FUNCTION_BLOCK FB_Fahrleitsystem
VAR_INPUT
END_VAR
VAR_OUTPUT
END_VAR
VAR
	Done : BOOL;
	Busy	: BOOL;
	Error : BOOL;
	StartStockwerk:	INT;
	ZielStockwerk:	INT;
	SicherheitsCheckbestanden : BOOL;
	AmStartStockwerk : BOOL;
	AmZielStockwerk : BOOL;
	TuerenZu : BOOL;
	Start : BOOL;
	AktuellesStockwerk : INT;
	Fahrauftragverstanden : BOOL;
	Tuerauftragverstanden : BOOL;
	State: ENUM_Fahrsystem;
	fbTuer : FB_Tuer;
	fbAchse : FB_Achse;
	AbholungFertig : BOOL;
	Closingdoors: BOOL;
	Achsereferenziert: BOOL;
	AufstartenAbgeschlossen : BOOL;
	AufstartenFreigabe : BOOL;
	AllDoorsClosed : BOOL;
	fbBlinker : FB_Blinker;
	FehlerQuittierenFlanke : R_TRIG;   // NEU — Flanke für Quittierung
 	sFehlertext : STRING(500);  // lokale Hilfsvariable
    i_txt       : INT;
END_VAR

fbAchse(Simulation:= , S_Zielposition:= , Achse:= IO_L1.LiftAxis);
fbTuer(
    SensorOpen1 := IO_L1.Door_1_SensorOpen,
    SensorOpen2 := IO_L1.Door_2_SensorOpen,
    SensorOpen3 := IO_L1.Door_3_SensorOpen,
    SensorOpen4 := IO_L1.Door_4_SensorOpen,
    SensorOpen5 := IO_L1.Door_5_SensorOpen,
    SensorOpen6 := IO_L1.Door_6_SensorOpen,

    SensorClosed1 := IO_L1.Door_1_SensorClosed,
    SensorClosed2 := IO_L1.Door_2_SensorClosed,
    SensorClosed3 := IO_L1.Door_3_SensorClosed,
    SensorClosed4 := IO_L1.Door_4_SensorClosed,
    SensorClosed5 := IO_L1.Door_5_SensorClosed,
    SensorClosed6 := IO_L1.Door_6_SensorClosed,

    Lichtschranke1 := IO_L1.Door_1_SensorActive,
    Lichtschranke2 := IO_L1.Door_2_SensorActive,
    Lichtschranke3 := IO_L1.Door_3_SensorActive,
    Lichtschranke4 := IO_L1.Door_4_SensorActive,
    Lichtschranke5 := IO_L1.Door_5_SensorActive,
    Lichtschranke6 := IO_L1.Door_6_SensorActive,

    MotorOpen1 => IO_L1.Door_1_MotorOpen,
    MotorOpen2 => IO_L1.Door_2_MotorOpen,
    MotorOpen3 => IO_L1.Door_3_MotorOpen,
    MotorOpen4 => IO_L1.Door_4_MotorOpen,
    MotorOpen5 => IO_L1.Door_5_MotorOpen,
    MotorOpen6 => IO_L1.Door_6_MotorOpen,

    MotorClose1 => IO_L1.Door_1_MotorClose,
    MotorClose2 => IO_L1.Door_2_MotorClose,
    MotorClose3 => IO_L1.Door_3_MotorClose,
    MotorClose4 => IO_L1.Door_4_MotorClose,
    MotorClose5 => IO_L1.Door_5_MotorClose,
    MotorClose6 => IO_L1.Door_6_MotorClose,
	AllDoorsClosed => AllDoorsClosed,
	FehlerQuittieren := IO_L1.Control_Reset
);

fbBlinker(bEnable:= TRUE, tOn:= T#500MS, tOff:=T#500MS , bOut=> );
SicherheitsCheckbestanden := FALSE;
Done := FALSE;
CASE State OF


	ENUM_Fahrsystem.Warten:
		Busy := FALSE;
		Done := FALSE;
		IF NOT 	AufstartenAbgeschlossen  AND IO_L1.Control_Automatic THEN
			Busy := TRUE;
			State := ENUM_Fahrsystem.Aufstartablauf;
		END_IF
		IF Start AND Divers.AutomatikmodusAktiv THEN
			Busy := TRUE;
			Start := FALSE;
			State := ENUM_Fahrsystem.Sicherheitscheck;
		END_IF
 		IF Visu_Manuellmodus.PosAnfahren AND Divers.ManuellmodusAktiv THEN
			ZielStockwerk := Visu_Manuellmodus.Zielstock;
 			State := ENUM_Fahrsystem.ZumZielStockwerk; 
		END_IF
	ENUM_Fahrsystem.Sicherheitscheck:
		//IF fbTuer.M_AreDoorsClosed() AND NOT fbAchse.M_isBusy() AND NOT fbAchse.M_hasError() THEN
			SicherheitsCheckbestanden := TRUE;
		//END_IF
		IF SicherheitsCheckbestanden THEN
			IF StartStockwerk = AktuellesStockwerk THEN
				State := ENUM_Fahrsystem.ZumZielStockwerk;
			END_IF
			IF StartStockwerk <> AktuellesStockwerk THEN 
				State := ENUM_Fahrsystem.ZumStartStockwerk;
			END_IF
		END_IF
		
	ENUM_Fahrsystem.Tueren:
		Busy := TRUE;	
		IF NOT Tuerauftragverstanden AND NOT fbAchse.M_isBusy() AND NOT fbAchse.M_hasError()THEN
			Tuerauftragverstanden := fbTuer.M_Tuerablaufstarten(AktuellesStockwerk);
		END_IF
		IF fbTuer.M_DoorOpen() THEN
			AbholungFertig := TRUE;
		ELSE 
			AbholungFertig := FALSE;
		END_IF
		IF fbTuer.M_isDone() THEN
			AbholungFertig := FALSE;
			Tuerauftragverstanden := FALSE;
			IF AmStartStockwerk THEN
				State := ENUM_Fahrsystem.ZumZielStockwerk;
			END_IF
			IF AmZielStockwerk THEN
				Done := TRUE; 
				State := ENUM_Fahrsystem.Warten;
			END_IF
		END_IF
	ENUM_Fahrsystem.ZumStartStockwerk:
		Busy := TRUE;
		AmZielStockwerk := FALSE;
		Fahrauftragverstanden := fbAchse.M_Movetoposition(StartStockwerk);
		IF fbAchse.M_isDone() THEN
			//OrderID_Counter.AktuellesStockwerk := StartStockwerk;
			AktuellesStockwerk := StartStockwerk;
			AmStartStockwerk := TRUE;
			State := ENUM_Fahrsystem.Tueren;
		END_IF
	ENUM_Fahrsystem.ZumZielStockwerk:
		Busy := TRUE;
		AmStartStockwerk := FALSE;
		Fahrauftragverstanden := fbAchse.M_Movetoposition(ZielStockwerk);
		IF fbAchse.M_isDone() THEN
			//OrderID_Counter.AktuellesStockwerk := ZielStockwerk;
			AktuellesStockwerk := ZielStockwerk;
			AmZielStockwerk := TRUE;
			IF Divers.AutomatikmodusAktiv THEN
				State := ENUM_Fahrsystem.Tueren;
			ELSE
				State := ENUM_Fahrsystem.Warten;	
			END_IF
			
		END_IF
	
	ENUM_Fahrsystem.Aufstartablauf: 
	Busy := TRUE;
	IF IO_L1.Control_Start THEN
		AufstartenFreigabe := TRUE;
	END_IF
		IF AufstartenFreigabe THEN
	
			IF NOT AllDoorsClosed THEN
				IO_L1.Control_LED_White := TRUE;
				Closingdoors := fbTuer.M_closeAllDoors();
			END_IF
			IF AllDoorsClosed THEN
				IO_L1.Control_LED_Red := TRUE;
				Achsereferenziert := fbAchse.M_Movetoposition(1);
					IF fbAchse.M_isDone() THEN
						AktuellesStockwerk := 1;
						AufstartenAbgeschlossen := TRUE;
						AufstartenFreigabe := FALSE;
						State := ENUM_Fahrsystem.Warten;
				END_IF
			END_IF
			
		END_IF
		
END_CASE


//LED Stuerung
IF IO_L1.Control_Automatic AND AufstartenAbgeschlossen THEN
    // Anlage läuft (mit oder ohne Auftrag) → dauernd an
    IO_L1.Control_LED_White := TRUE;

ELSIF IO_L1.Control_Automatic AND NOT AufstartenAbgeschlossen THEN
    // Aufstartablauf → blinken
    IO_L1.Control_LED_White := fbBlinker.bOut;

ELSIF NOT IO_L1.Control_Automatic AND Busy THEN
    // Automatik verlassen, Auftrag wird noch fertig gemacht → blinken
    IO_L1.Control_LED_White := fbBlinker.bOut;

ELSE
    // Kein Automatik, kein aktiver Auftrag → aus
    IO_L1.Control_LED_White := FALSE;
END_IF
// ── Fehler sammeln ────────────────────────────────────────────────────────────
Divers.Fehler.AchsePower := fbAchse.fbPower.Error;
Divers.Fehler.AchseHome  := fbAchse.fbHome.Error;
Divers.Fehler.AchseMove  := fbAchse.fbMoveAbs.Error;
Divers.Fehler.AchseJog   := fbAchse.fbJog.Error;
Divers.Fehler.NotAus     := IO_L1.Control_EmergencyStopActive;
Divers.Fehler.TuerTimeout := fbTuer.TuerFehler;

// Letzten Achsen-Fehlercode speichern
IF fbAchse.fbPower.Error   THEN Divers.Fehler.AchseFehlercode := fbAchse.FehlercodePower; END_IF
IF fbAchse.fbHome.Error    THEN Divers.Fehler.AchseFehlercode := fbAchse.FehlercodeRef;   END_IF
IF fbAchse.fbMoveAbs.Error THEN Divers.Fehler.AchseFehlercode := fbAchse.FehlercodeMove;  END_IF

// Zusammenfassung
Divers.Fehler.IrgendeinFehler :=
    Divers.Fehler.AchsePower OR
    Divers.Fehler.AchseHome  OR
    Divers.Fehler.AchseMove  OR
    Divers.Fehler.AchseJog   OR
    Divers.Fehler.NotAus     OR
    Divers.Fehler.TuerTimeout[1] OR Divers.Fehler.TuerTimeout[2] OR
    Divers.Fehler.TuerTimeout[3] OR Divers.Fehler.TuerTimeout[4] OR
    Divers.Fehler.TuerTimeout[5] OR Divers.Fehler.TuerTimeout[6];

Divers.Fehler.IrgendEineWarnung := IO_L1.Control_Overload;

// ── Quittierung ───────────────────────────────────────────────────────────────
FehlerQuittierenFlanke(CLK := IO_L1.Control_Reset);
IF FehlerQuittierenFlanke.Q AND NOT Divers.Fehler.IrgendeinFehler THEN
    Divers.Fehler.FehlerQuittiert := TRUE;
END_IF
IF Divers.Fehler.IrgendeinFehler THEN
    Divers.Fehler.FehlerQuittiert := FALSE;  // Reset bei neuem Fehler
END_IF

// ── LED Steuerung Rot / Blau / Gelb ──────────────────────────────────────────
IF Divers.Fehler.IrgendeinFehler THEN
    IO_L1.Control_LED_Red := TRUE;
    IF Divers.Fehler.FehlerQuittiert THEN
        IO_L1.Control_LED_Blue := fbBlinker.bOut;  // blinkt = quittierbar
    ELSE
        IO_L1.Control_LED_Blue := TRUE;             // dauernd = noch aktiv
    END_IF
ELSE
    IO_L1.Control_LED_Red  := FALSE;
    IO_L1.Control_LED_Blue := FALSE;
END_IF

IO_L1.Control_LED_Yellow := Divers.Fehler.IrgendEineWarnung;
// ─────────────────────────────────────────────────────────────────────────────
// ── Fehlertext aufbauen ───────────────────────────────────────────────────────
sFehlertext := '';

// Achse
IF Divers.Fehler.AchsePower THEN
    sFehlertext := CONCAT(sFehlertext, 'FEHLER: Achse Power');
    sFehlertext := CONCAT(sFehlertext, CONCAT(' (Code: ', CONCAT(UDINT_TO_STRING(Divers.Fehler.AchseFehlercode), ') | ')));
END_IF
IF Divers.Fehler.AchseHome THEN
    sFehlertext := CONCAT(sFehlertext, 'FEHLER: Referenzfahrt');
    sFehlertext := CONCAT(sFehlertext, CONCAT(' (Code: ', CONCAT(UDINT_TO_STRING(Divers.Fehler.AchseFehlercode), ') | ')));
END_IF
IF Divers.Fehler.AchseMove THEN
    sFehlertext := CONCAT(sFehlertext, 'FEHLER: Positionierung');
    sFehlertext := CONCAT(sFehlertext, CONCAT(' (Code: ', CONCAT(UDINT_TO_STRING(Divers.Fehler.AchseFehlercode), ') | ')));
END_IF
IF Divers.Fehler.AchseJog THEN
    sFehlertext := CONCAT(sFehlertext, 'FEHLER: Jog | ');
END_IF

// Türen
FOR i_txt := 1 TO 6 DO
    IF Divers.Fehler.TuerTimeout[i_txt] THEN
        sFehlertext := CONCAT(sFehlertext, 'FEHLER: Tuer Timeout Stock. ');
        sFehlertext := CONCAT(sFehlertext, CONCAT(INT_TO_STRING(i_txt), ' | '));
    END_IF
END_FOR

// Allgemein
IF Divers.Fehler.NotAus THEN
    sFehlertext := CONCAT(sFehlertext, 'FEHLER: Not-Aus | ');
END_IF
IF Divers.Fehler.Brandalarm THEN
    sFehlertext := CONCAT(sFehlertext, 'FEHLER: Brandalarm | ');
END_IF

// Warnung
IF Divers.Fehler.IrgendEineWarnung THEN
    sFehlertext := CONCAT(sFehlertext, 'WARNUNG: Ueberlast Kabine | ');
END_IF

// Kein Fehler
IF sFehlertext = '' THEN
    sFehlertext := 'Keine Fehler';
END_IF

Divers.Fehlertext := sFehlertext;
// ─────────────────────────────────────────────────────────────────────────────

METHOD PUBLIC M_AbholungFertig : INT
VAR_INPUT
END_VAR
IF AbholungFertig THEN
	M_AbholungFertig := ZielStockwerk;
ELSE
	M_AbholungFertig := -1;
END_IF
END_METHOD

METHOD PUBLIC M_AcceptTask : BOOL
VAR_INPUT
Task : ST_Fahrauftrag;

END_VAR
IF NOT Busy THEN
	StartStockwerk := Task.Startstockwerk;
	Zielstockwerk := Task.Zielstockwerk;
	Start:= TRUE;
	M_AcceptTask := TRUE;
ELSE 
	M_AcceptTask := FALSE;
END_IF
END_METHOD

METHOD PUBLIC M_isBusy : BOOL
VAR_INPUT
END_VAR
M_isBusy := Busy;
END_METHOD

METHOD PUBLIC M_isDone : BOOL
VAR_INPUT
END_VAR
M_isDone := Done;
END_METHOD

END_FUNCTION_BLOCK

(* stored: Version 1.1.0.1
   POU FB_Fahrleitsystem: Id {7583cd05-68d7-4c93-9869-d2e80ddd0766}, SpecialFunc None
   Method M_AbholungFertig: Id {d534390c-596d-410a-950e-73e20c0959ce}
   Method M_AcceptTask: Id {d5baa6a5-1e56-45e8-ab59-264b78e34233}
   Method M_isBusy: Id {d1622e40-44df-4c6b-903a-d2cb1245845e}
   Method M_isDone: Id {12d4a25e-6ae5-44be-a9c4-3f89ee142147} *)
